// TIA Portal project "Project5" (V15)
// Vorlageprojekt für das Buch mit Zielsystem S7-1200

(* hardware
DEVICE "S7-1200-Station_1"  S7-1200 Station
   slot 0: "Baugruppenträger_0"  Rack  V1.0
   slot 1: "PLC_1"  CPU 1211C DC/DC/DC  6ES7 211-1AE40-0XB0  V4.1
*)

// ===== PLC "PLC_1"  CPU 1211C DC/DC/DC =====

VAR_GLOBAL   // PLC tag table "Standard-Variablentabelle"
   "START" AT %I0.0 : Bool;
   "STOP" AT %I0.1 : Bool;
   "Selector 1" AT %I0.2 : Bool;
   "Selector 2" AT %I0.3 : Bool;
   "S FRONT LIMIT" AT %I0.5 : Bool;
   "BELT 4m" AT %Q0.0 : Bool;
   "PUSHER" AT %Q0.1 : Bool;
   "X" AT %M0.0 : Bool;
   "S BACK LIMIT" AT %I0.4 : Bool;
   "SENSOR 1" AT %I0.6 : Bool;
   "SENSOR 2" AT %I0.7 : Bool;
   "Tag_1" AT %M1.0 : Bool;
   "Tag_2" AT %M1.1 : Bool;
   "Tag_3" AT %M1.5 : Bool;
   "Tag_4" AT %M1.4 : Bool;
   "Tag_5" AT %M1.6 : Bool;
   "Y" AT %M0.1 : Bool;
   "Tag_6" AT %M0.5 : Bool;
END_VAR

FUNCTION "MHJ-PLC-Lab-Function-S71200" : Void   // FC9000, SCL
{ S7_Optimized_Access := 'TRUE' }
VERSION : 0.1
   VAR_TEMP
      rdTimeReturn : Int;
      outputTime : DTL;
      SyncVal : Byte;
      forVal : Int;
      forVal_2 : Int;
      Value : Byte;
   END_VAR
   VAR CONSTANT
      CompVal : Byte := 16#34;
      Value_01 : Byte := 16#11;
      Value_01_DW : DWord := 16#A165_D992;
      Value_02_DW : DWord := 16#58BE_4401;
   END_VAR
BEGIN

   #Value:=PEEK(area := 16#82,
        dbNumber := 0,
        byteOffset := 511);
   #Value := #Value + 1;

   POKE(area := 16#82,
        dbNumber := 0,
        byteOffset := 511,
        value := #Value);

   POKE(area:=16#81,
        dbNumber:=0,
        byteOffset:=1016,
        value:=#Value_01_DW);
   POKE(area := 16#81,
        dbNumber := 0,
        byteOffset := 1020,
        value := #Value_02_DW);

   POKE(area := 16#81,
        dbNumber := 0,
        byteOffset := 511,
        value := B#16#00);

   FOR #forVal := 0 TO 120 DO
       FOR #forVal_2:=0 TO 10 DO
           #rdTimeReturn:=RD_SYS_T(#outputTime);
           #rdTimeReturn := WR_SYS_T(#outputTime);
           #rdTimeReturn := RD_SYS_T(#outputTime);
           #rdTimeReturn := WR_SYS_T(#outputTime);
       END_FOR;
       #SyncVal:= PEEK(area := 16#81,
                      dbNumber := 0,
                      byteOffset := 511);
       IF #SyncVal = #CompVal THEN
          GOTO M_1;
       END_IF;
   END_FOR;
   RETURN;

   M_1:
   POKE(area := 16#81,
        dbNumber := 0,
        byteOffset := 511,
        value := B#16#0);
END_FUNCTION

ORGANIZATION_BLOCK "Main"   // OB1, LAD, ProgramCycle
TITLE = "Main Program Sweep (Cycle)"
{ S7_Optimized_Access := 'TRUE' }
VERSION : 0.1
   VAR_INPUT
      Initial_Call : Bool;   // Initial call of this OB
      Remanence : Bool;   // =True, if remanent data are available
   END_VAR
   VAR_TEMP   // added for the SCL form of the ladder/FBD networks
      _w1 : Bool;
      _w2 : Bool;
      _w3 : Bool;
   END_VAR
BEGIN

REGION Network 1: Konnektierungsbaustein für PLC-Lab
   // Im Netzwerk 1 wird der Konnektierungsbaustein für PLC-Lab aufgerufen.
   // Dieser Aufruf darf nicht entfernt werden!
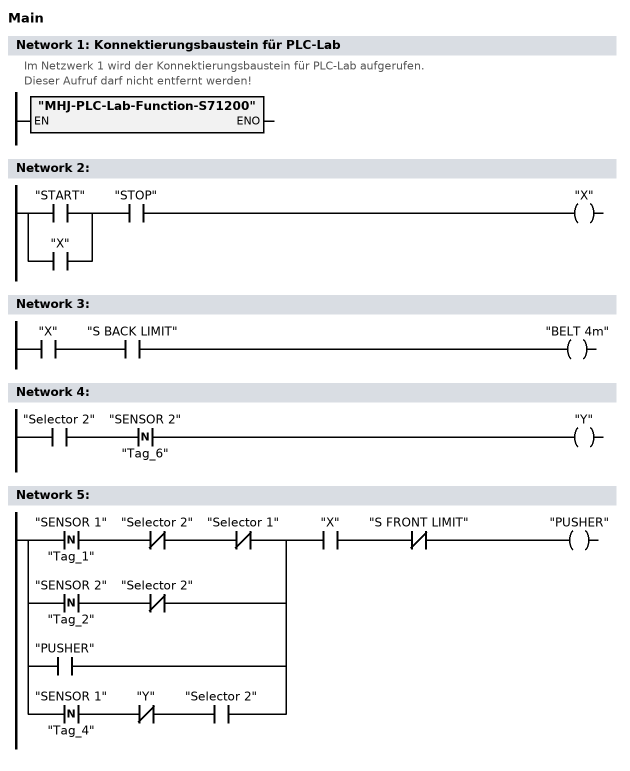
   RUNG wire#powerrail
      "MHJ-PLC-Lab-Function-S71200"()
   END_RUNG
   // the same network as SCL:
   "MHJ-PLC-Lab-Function-S71200"();
END_REGION

REGION Network 2
   RUNG wire#powerrail
      Contact( "START" )
      wire#w1
      Contact( "STOP" )
      Coil( "X" )
   END_RUNG
   RUNG wire#powerrail
      Contact( "X" )
   END_RUNG wire#w1
   // the same network as SCL:
   "X" := ("START" OR "X") AND "STOP";
END_REGION

REGION Network 3
   RUNG wire#powerrail
      Contact( "X" )
      Contact( "S BACK LIMIT" )
      Coil( "BELT 4m" )
   END_RUNG
   // the same network as SCL:
   "BELT 4m" := "X" AND "S BACK LIMIT";
END_REGION

REGION Network 4
   RUNG wire#powerrail
      Contact( "Selector 2" )
      N_Contact(operand := "SENSOR 2", bit := "Tag_6")
      Coil( "Y" )
   END_RUNG
   // the same network as SCL:
   #_w1 := "Selector 2" AND NOT "SENSOR 2" AND "Tag_6";   // falling edge of "SENSOR 2"
   "Tag_6" := "SENSOR 2";
   "Y" := #_w1;
END_REGION

REGION Network 5
   RUNG wire#powerrail
      N_Contact(operand := "SENSOR 1", bit := "Tag_1")
      I_Contact( "Selector 2" )
      I_Contact( "Selector 1" )
      wire#w1
      Contact( "X" )
      I_Contact( "S FRONT LIMIT" )
      Coil( "PUSHER" )
   END_RUNG
   RUNG wire#powerrail
      N_Contact(operand := "SENSOR 2", bit := "Tag_2")
      I_Contact( "Selector 2" )
   END_RUNG wire#w1
   RUNG wire#powerrail
      Contact( "PUSHER" )
   END_RUNG wire#w1
   RUNG wire#powerrail
      N_Contact(operand := "SENSOR 1", bit := "Tag_4")
      I_Contact( "Y" )
      Contact( "Selector 2" )
   END_RUNG wire#w1
   // the same network as SCL:
   #_w1 := NOT "SENSOR 1" AND "Tag_1";   // falling edge of "SENSOR 1"
   "Tag_1" := "SENSOR 1";
   #_w2 := NOT "SENSOR 2" AND "Tag_2";   // falling edge of "SENSOR 2"
   "Tag_2" := "SENSOR 2";
   #_w3 := NOT "SENSOR 1" AND "Tag_4";   // falling edge of "SENSOR 1"
   "Tag_4" := "SENSOR 1";
   "PUSHER" := ((#_w1 AND NOT "Selector 2" AND NOT "Selector 1") OR (#_w2 AND NOT "Selector 2") OR "PUSHER" OR (#_w3 AND NOT "Y" AND "Selector 2")) AND "X" AND NOT "S FRONT LIMIT";
END_REGION
END_ORGANIZATION_BLOCK